TEXTLIST TextList_Orders
  0 = 'open' | FR: 'Ouvrir' | EN: 'Open'
  1 = 'close' | FR: 'Fermer' | EN: 'Close'
  2 = 'Clampage' | FR: 'Clampage' | EN: 'Clamping'
  3 = 'Déclampage' | FR: 'Déclampage' | EN: 'Unclamping'
   = ''
END_TEXTLIST

(* stored: Version 1.1.0.1, ProductVersion 3.1.4024.10
   TextList TextList_Orders: Id {e7423938-72dd-44f3-bca9-eabc69ec25ec} *)
